(* PLC project Unnamed, Unknown Unnamed 1 *)
(* stored: creationDateTime 2022-08-18T16:52:56, modificationDateTime 2022-08-19T23:55:26 *)

PROGRAM Traffic_Control
  VAR_INPUT
    Start_PB : BOOL := FALSE;
    Stop_PB : BOOL := FALSE;
    Pedestrian_PB : BOOL := FALSE;
  END_VAR
  VAR
    STEP0_Action : BOOL := FALSE;
    STEP0_1Action : BOOL := FALSE;
    STEP1_Action : BOOL := FALSE;
    STEP2_Action : BOOL := FALSE;
    RED_Light : BOOL := FALSE;
    YELLOW_Light : BOOL := FALSE;
    GREEN_Light : BOOL := FALSE;
    TON0 : TON;
    TON0_1 : TON;
    TON1 : TON;
    TON2 : TON;
    R_TRIG0 : R_TRIG;
  END_VAR
  VAR  (* added by the conversion: wires and edge detectors of the diagram *)
    _OR20_OUT : BOOL;
  END_VAR

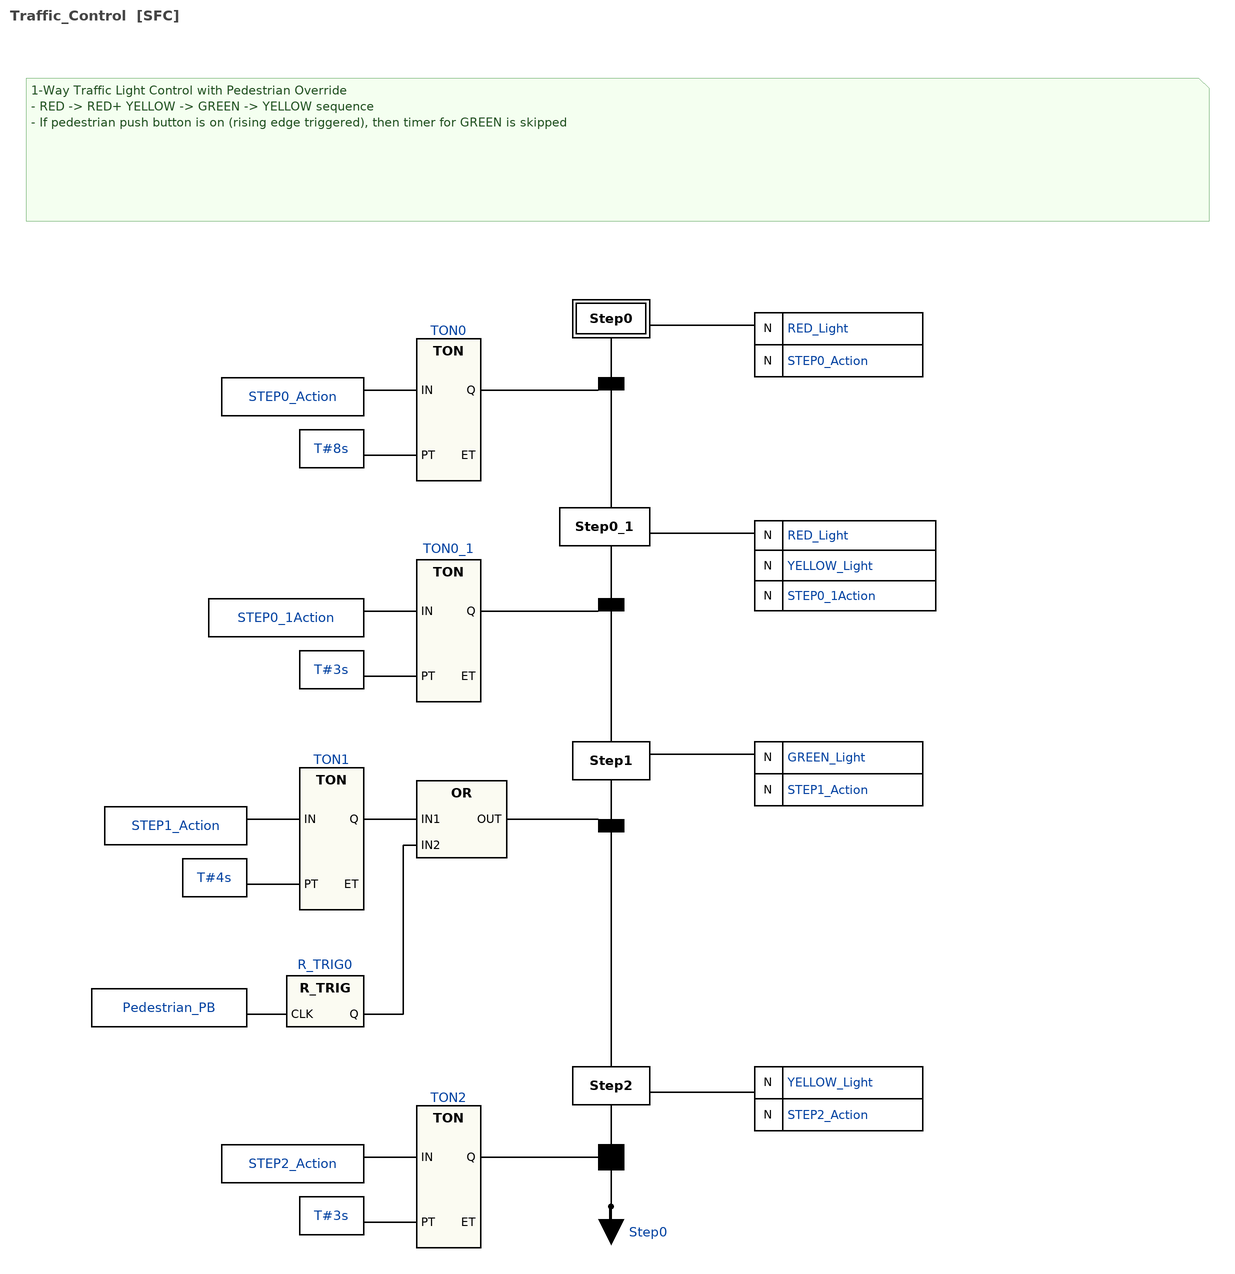
(* 1-Way Traffic Light Control with Pedestrian Override
- RED -> RED+ YELLOW -> GREEN -> YELLOW sequence
- If pedestrian push button is on (rising edge triggered), then timer for GREEN is skipped *)
INITIAL_STEP Step0:
  RED_Light(N);
  STEP0_Action(N);
  COMPUTE_FUNCTION_BLOCKS(S);
END_STEP
TRANSITION FROM Step0 TO Step0_1
  := TON0.Q;
END_TRANSITION
STEP Step0_1:
  RED_Light(N);
  YELLOW_Light(N);
  STEP0_1Action(N);
END_STEP
TRANSITION FROM Step0_1 TO Step1
  := TON0_1.Q;
END_TRANSITION
STEP Step1:
  GREEN_Light(N);
  STEP1_Action(N);
END_STEP
TRANSITION FROM Step1 TO Step2
  := _OR20_OUT;
END_TRANSITION
STEP Step2:
  YELLOW_Light(N);
  STEP2_Action(N);
END_STEP
TRANSITION FROM Step2 TO Step0
  := TON2.Q;
END_TRANSITION
ACTION COMPUTE_FUNCTION_BLOCKS:  (* blocks drawn on the SFC sheet *)
  TON0(IN := STEP0_Action, PT := T#8s);
  TON0_1(IN := STEP0_1Action, PT := T#3s);
  TON1(IN := STEP1_Action, PT := T#4s);
  R_TRIG0(CLK := Pedestrian_PB);
  _OR20_OUT := TON1.Q OR R_TRIG0.Q;
  TON2(IN := STEP2_Action, PT := T#3s);
END_ACTION
END_PROGRAM

CONFIGURATION Config0
  RESOURCE Res0 ON PLC
    TASK task0(INTERVAL := T#20ms, PRIORITY := 0);
    PROGRAM instance0 WITH task0 : Traffic_Control;
  END_RESOURCE
END_CONFIGURATION
